// TIA Portal V19 export
TYPE "LAF_typeOperationInterlockCommands"
TITLE = LLGES_OperatorInterlockCommands
// Module related commands from external systems
// stored: Access Published
   STRUCT
      reqMaintenanceLock : Bool;   // TRUE: Request maintenance lock from HMI
      reqMaintenanceReset : Bool;   // TRUE: Request reset of maintenance lock from HMI
      serverMachineName : WString := WSTRING#'DEFAULT';   // @ServerMachineName tag of the panel currently in Operation
      localMachineName : WString := WSTRING#'DEFAULT';
   END_STRUCT;
END_TYPE
